FUNCTION_BLOCK FB_HydrualicSystem EXTENDS StateMachineBase
VAR_INPUT
    bIsSimulator : BOOL;

	// Hydrualic pump
	bHasPump : BOOL;
	sTypeOfPump : STRING;

	// Pressure sensor
	bHasPressureSensor : BOOL;
	sTypeOfPressureSensor : STRING;

    PressureSensor_input : st_PressureTransducer_Input;
END_VAR
VAR_OUTPUT
    bBusy : BOOL;
    bError : BOOL;
    bDone : BOOL;
    
    hydrualicPump_output : ST_Pump_Output;

    PLCtoHMI : st_PLCtoHMI_Hydrualics;
END_VAR
VAR
	// Function block instances for Hydrualic Pump
	fbPumpRealy : FB_Pump_RelayOnly;
	fbPumpHPU : FB_Pump_HPU;
    fbPumpSim : FB_Pump_Simulator;
    // Interface to pump
	iHydrualicPump : I_HydrualicPump;

    // Function block instances for Pressure Sensor
	fbPressureSensorSim : FB_PressureTransceiver_Sim;
	fbGenericPressureSensor : FB_GenericBrand_Transceiver;
    // Interface to Pressure Sensor
	iPressureSensor : I_PressureSensor;

    PressureValueMem : LREAL;

    primePumpTimeoutTON : TON := (PT := T#500ms);
    
END_VAR

M_VariantControl();
HandleInputs();

MonitorErrors();

ExecuteState();
IF NOT (nextState = curState) THEN
	StateTransition();
END_IF

fbPumpRealy();
fbPumpHPU();
fbPumpSim();
fbPressureSensorSim(simCellState := cellState);
fbGenericPressureSensor();

HandleOutputs();

ACTION ExecuteState:


CASE curState OF
	eState_Idle: ExecuteState_Idle();
	eState_Startup: ExecuteState_Startup();
	eState_Running: ExecuteState_Running();
	eState_Complete: ExecuteState_Complete();
	eState_Error: ExecuteState_Error();
	eState_Independent: ExecuteState_Independent();
END_CASE
END_ACTION

ACTION ExecuteState_Complete:

END_ACTION

ACTION ExecuteState_Error:

// stop pump in case of error
IF NOT (iHydrualicPump.getState() = eState_Idle) AND NOT (iHydrualicPump.getState() = eState_Error) THEN
    iHydrualicPump.stop();
END_IF
END_ACTION

ACTION ExecuteState_Idle:

END_ACTION

ACTION ExecuteState_Independent:

END_ACTION

ACTION ExecuteState_Running:
// I would setup every type of control loop here in a case statemant
// here I'm only using one (bang bang) as what is there to control with just ON/OFF

IF iPressureSensor.getSignal() > 10 THEN
    nextState := eState_Error;
    // throw overpressure error
    RETURN;
END_IF

// bang bang control
IF iPressureSensor.getSignal() > 9.9 THEN
    IF NOT (iHydrualicPump.getState() = eState_Idle) THEN
        // stop once pressure is above set point
        iHydrualicPump.stop();
    END_IF
ELSIF iPressureSensor.getSignal() <= 8.2 THEN
    IF NOT (iHydrualicPump.getState() = eState_Running) THEN
        // start once pressure below minimun
        iHydrualicPump.start();
    END_IF
END_IF
END_ACTION

ACTION ExecuteState_Startup:

IF (iHydrualicPump.getState() = eState_Idle) AND NOT (iHydrualicPump.getState() = eState_Error) THEN
    iHydrualicPump.start();
ELSE
    // failed to start error
END_IF

IF iPressureSensor.getSignal() > 8 THEN
    nextState := eState_Running;
END_IF

primePumpTimeoutTON(IN := (PressureValueMem > iPressureSensor.getSignal()));
IF primePumpTimeoutTON.Q THEN
    // failed to pressureize system. Checks for leaks! Or faulty motor.
    nextState := eState_Error;
END_IF

IF iPressureSensor.getSignal() > PressureValueMem THEN
    PressureValueMem := iPressureSensor.getSignal();
END_IF
END_ACTION

METHOD HandleInputs : BOOL
VAR_INPUT
END_VAR

// Pass pressure value to iPressureSensor
IF bIsSimulator THEN
    // pass pump state back to pressure sensor to generate sim signal
    fbPressureSensorSim.bPumpIsON := iHydrualicPump.getState() = eState_Running;
ELSE
    iPressureSensor.setSignal(PressureSensor_input.value);    
END_IF
END_METHOD

METHOD HandleOutputs : BOOL
VAR_INPUT
END_VAR
// Set Outputs
hydrualicPump_output.On := iHydrualicPump.getSignal();

// populate HMI struct
PLCtoHMI.state := curState;
PLCtoHMI.psiSensor.value := iPressureSensor.getSignal();
PLCtoHMI.pump.state := iHydrualicPump.getState();
END_METHOD

METHOD PRIVATE M_VariantControl : BOOL
VAR_INPUT
END_VAR
// Handle hydrualic pump options
IF bIsSimulator THEN
    iHydrualicPump := fbPumpSim;
    iPressureSensor := fbPressureSensorSim;
ELSE
    IF sTypeOfPump='relay' THEN
        iHydrualicPump := fbPumpRealy;
    ELSIF sTypeOfPump='hpu' THEN
        iHydrualicPump := fbPumpHPU;
    ELSE
        iHydrualicPump := fbPumpRealy;
    END_IF
    
    iPressureSensor := fbGenericPressureSensor;
END_IF
END_METHOD

METHOD MonitorErrors : BOOL
VAR_INPUT
END_VAR
// error if hydrualic pump fails
IF iHydrualicPump.getState() = eState_Error THEN
    nextState := eState_Error;
    // throw pump error
END_IF

IF curState = eState_Running THEN
    IF iPressureSensor.getSignal() < 8 THEN
        iHydrualicPump.stop();
        nextState := eState_Error;
        // throw pressure drop error
    END_IF
END_IF
END_METHOD

METHOD reset : BOOL
resetAlarms();

iHydrualicPump.reset();

nextState := eState_Idle;
END_METHOD

METHOD start: BOOL
VAR_INPUT
END_VAR
IF curState = eState_Idle THEN
	nextState := eState_Startup;
	start := TRUE;
ELSE
	start := FALSE;
END_IF
END_METHOD

ACTION StateTransition:
//reset timers


IF nextState = eState_Startup THEN
	primePumpTimeoutTON(IN := FALSE);
    PressureValueMem := iPressureSensor.getSignal();
END_IF


SUPER^.StateTransition();
END_ACTION

END_FUNCTION_BLOCK

(* stored: Version 1.1.0.1, ProductVersion 3.1.4024.9
   POU FB_HydrualicSystem: Id {480141df-1e34-4c40-90c2-d984119b85af}, SpecialFunc None
   Folder StateMachine: Id {551fd8e7-5396-43af-90e4-be09813ca759}
   Folder States: Id {71340a8b-6047-4c14-8703-c18cf8956771}
   Action ExecuteState: Id {60ea2387-7ca3-476e-9945-c00f184a2b15}
   Action ExecuteState_Complete: Id {775318d5-b27f-43fe-9655-bcf8367d2057}
   Action ExecuteState_Error: Id {9892b3ef-3084-45a8-bc26-fc6ac99458f2}
   Action ExecuteState_Idle: Id {dc8f3035-e716-4cb8-b759-a71852a0ee7e}
   Action ExecuteState_Independent: Id {dd7ece7a-48c8-4285-a849-c3868fe2a7df}
   Action ExecuteState_Running: Id {02225357-1a6b-41f2-8157-2082449ed525}
   Action ExecuteState_Startup: Id {d0702009-a7fe-4669-9e13-2151537efaff}
   Method HandleInputs: Id {c2b4d46f-73ad-4ab8-af7d-00bc44906398}
   Method HandleOutputs: Id {e3e17ff5-98c8-42eb-ad85-eeeacfd37523}
   Method M_VariantControl: Id {0c3baa99-c2be-4e7a-96b3-9ba353a2863b}
   Method MonitorErrors: Id {7052d4e8-391a-4e78-8109-17d9eadd25cb}
   Method reset: Id {b88535b0-eef6-46db-8072-184167fea706}
   Method start: Id {e488af84-cccf-49de-ae23-71c832f7a38a}
   Action StateTransition: Id {6d75eee6-daa0-4c71-9782-29847b401a73} *)
